Universal Robots URScript: movimientos.script

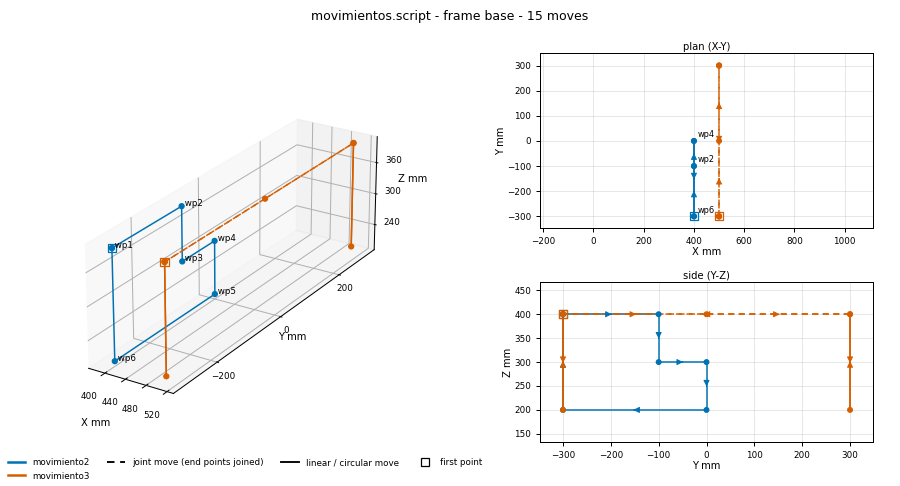
[picture p0: tool path of movimientos.script in frame base, 15 of 21 moves have a stored position in this frame; points joined in program order, loops and branches not executed]
def tarea1(tipo_oper, num_oper):

    cont_oper = 0
    while (cont_oper < num_oper):
        if tipo_oper == 1:
            movimiento1()
        elif tipo_oper == 2:
            movimiento2()https://prod.liveshare.vsengsaas.visualstudio.com / join?EEAD140651B9BF86DB2DEE8C123D3F0B23D8
        elif tipo_oper == 3:
            movimiento3()
        else:
            halt
        end
        cont_oper = cont_oper + 1
    end
end

def movimiento1():

    wp1r = get_actual_tcp_pose()
    wp2r = pose_trans(wp1r, p[0, 0.2, 0, 0, 0, 0])
    wp3r = pose_trans(wp2r, p[0, 0, 0.1, 0, 0, 0])
    wp4r = pose_trans(wp3r, p[0, 0.1, 0, 0, 0, 0])
    wp5r = pose_trans(wp4r, p[0, 0, 0.1, 0, 0, 0])
    wp6r = pose_trans(wp5r, p[0, -0.3, 0, 0, 0, 0])
    movel(wp2r)
    movel(wp3r)
    movel(wp4r)
    movel(wp5r)
    movel(wp6r)
    movel(wp1r)
    popup("Paso un ciclo", blocking = True)

end
def movimiento2():
    #Waypoints definidos por poses
    wp1 = p[0.4, -0.3, 0.4, 0, 1.57, 0]
    wp2 = p[0.4, -0.1, 0.4, 0, 1.57, 0]
    wp3 = p[0.4, -0.1, 0.3, 0, 1.57, 0]
    wp4 = p[0.4, 0, 0.3, 0, 1.57, 0]
    wp5 = p[0.4, 0, 0.2, 0, 1.57, 0]
    wp6 = p[0.4, -0.3, 0.2, 0, 1.57, 0]
    lpai = [-0.604, -1.204, -2.091, -1.417, 1.569, 0]

    #Movimientos
    movej(get_inverse_kin(wp1, qnear = lpai))
    movel(wp2, r = 0.05)
    movel(wp3, r = 0.05)
    movel(wp4, r = 0.05)
    movel(wp5)
    movel(wp6, r = 0.05)
    movel(wp1)
end

def movimiento3():
    #Waypoints guardados como poses
    wp1 = p[0.5, -0.3, 0.4, 0, 3.14, 0]
    wp2 = p[0.5, -0.3, 0.2, 0, 3.14, 0]
    wp3 = p[0.5, 0, 0.4, 0, 3.14, 0]
    wp4 = p[0.5, 0.3, 0.4, 0, 3.14, 0]
    wp5 = p[0.5, 0.3, 0.2, 0, 3.14, 0]
    lpai = [-0.604, -1.204, -2.091, -1.417, 1.569, 0]

    #Movimientos
    movej(get_inverse_kin(wp1, qnear = lpai))

    movel(wp2)
    movel(wp1)

    movej(get_inverse_kin(wp3))
    popup("Continue cuando el proceso haya acabado", title = "¿Ya acabo el proceso?", blocking = True)
    movej(get_inverse_kin(wp4))

    movel(wp5)
    movel(wp4)

    movej(get_inverse_kin(wp1, qnear = lpai))
end
